// TIA Portal V20 export
TYPE "LER_typeCommunicationCommands"
// stored: Access Published
   STRUCT
      Communication_Reset { S7_SetPoint := 'True'} : Bool;
   END_STRUCT;
END_TYPE
